// TIA Portal project "ForExportDB" (V14)

(* hardware
DEVICE "S7300/ET200M station_1"  S7-300 station
   slot 0: "Rail_0"  Rail  6ES7 390-1***0-0AA0
   slot 2: "PLC_1"  CPU 315-2 PN/DP  6ES7 315-2EH14-0AB0  V3.2
      slot 2: "PROFINET interface_1"  PN-IO
         slot 1: "Port_1"  Port
         slot 2: "Port_2"  Port
*)

// ===== PLC "PLC_1"  CPU 315-2 PN/DP =====

TYPE "UDT_DESCRETE_MODULE"
   STRUCT
      D_0 : Bool;
      D_1 : Bool;
      D_2 : Bool;
      D_3 : Bool;
      D_4 : Bool;
      D_5 : Bool;
      D_6 : Bool;
      D_7 : Bool;
      xEmpty : Bool;
      bByte : Byte;
   END_STRUCT;
END_TYPE

TYPE "UDT_FLOWRATE_PULSE"
   STRUCT
      iPulseCounter : Int;   // Счетчик импульсов
      xResetCounter : Bool;   // Сброс счетчика
      rPulseFlowRate : Real;   // Расход
      rPulseRes : Real := 100.0;   // Сколько мл/л на импульс (100 мл / имп)
      rSumFlowPanel : Real;   // Суммарный расход всего
      rSumFlowProg : Real;   // Суммарный расход доза
      xResetFlowRateProg : Bool;   // Сброс СРВ
      xResetFlowRatePanel : Bool;   // Сброс СРД
   END_STRUCT;
END_TYPE

TYPE "UDT_ALARM"
   STRUCT
      LAMPS : Struct   // Индикация
         Lamp1 : Struct   // Светофор 1
            rFlashTimer : Real := 3.0;   // Значение мигания
            iLampState : Array[0..2] of Int;   // Режим работы ламп
            xLampFlash : Array[0..2] of Bool;   // Мигание включено или нет
            xLampSet : Array[0..2] of Bool;
         END_STRUCT;
         Lamp2 : Struct   // Светофор 2
            rFlashTimer : Real := 1.0;   // Значение мигания
            iLampState : Array[0..2] of Int;   // Режим работы ламп
            xLampFlash : Array[0..2] of Bool;   // Мигание включено или нет
            xLampSet : Array[0..2] of Bool;
         END_STRUCT;
         Panel : Struct   // Индикация на панели
            xBuzzer : Bool;   // Звук
            xStartLamp : Bool;   // Старт
            xStopLamp : Bool;   // Стоп
            xResetLamp : Bool;   // Сброс
         END_STRUCT;
         Stand : Struct   // Индикация на стенде
            xRunMotor : Bool;   // Лампа мотора
            rRunMotorFlashTime : Real := 2.0;   // Значение мигания
         END_STRUCT;
      END_STRUCT;
      STATUS : Struct   // Статусы
         xErrorCommon : Bool;   // Общая ошибка
         xWarningCommon : Bool;   // Общее предупреждение
         iWarning : Int;   // Слово состояние предупреждения
         iError : Int;   // Слово состояния ошибки
         bMode : Byte;   // Текущий режим работы системы 16#25-26-29-2A
      END_STRUCT;
   END_STRUCT;
   // LAMPS.Lamp1.xLampFlash[0] := TRUE;
   // LAMPS.Lamp1.xLampFlash[1] := TRUE;
   // LAMPS.Lamp1.xLampFlash[2] := TRUE;
   // LAMPS.Lamp2.xLampFlash[0] := FALSE;
   // LAMPS.Lamp2.xLampFlash[1] := TRUE;
   // LAMPS.Lamp2.xLampFlash[2] := FALSE;
   // LAMPS.Lamp1.iLampState[0] := 0;   // Режим работы ламп красный
   // LAMPS.Lamp1.iLampState[1] := 1;   // Режим работы ламп желтый
   // LAMPS.Lamp1.iLampState[2] := 2;   // Режим работы ламп зеленый
   // LAMPS.Lamp2.iLampState[0] := 2;   // Режим работы ламп красный
   // LAMPS.Lamp2.iLampState[1] := 1;   // Режим работы ламп желтый
   // LAMPS.Lamp2.iLampState[2] := 0;   // Режим работы ламп зеленый
END_TYPE

TYPE "UDT_ANALOG_AI_MODULE"
   STRUCT
      AI_0 : Struct
         RAW : "UDT_IO_ANALOG_M1";
         SCALE : "UDT_SCALE_AI";
      END_STRUCT;
      AI_1 : Struct
         RAW : "UDT_IO_ANALOG_M1";
         SCALE : "UDT_SCALE_AI";
      END_STRUCT;
      AI_2 : Struct
         RAW : "UDT_IO_ANALOG_M1";
         SCALE : "UDT_SCALE_AI";
      END_STRUCT;
      AI_3 : Struct
         RAW : "UDT_IO_ANALOG_M1";
         SCALE : "UDT_SCALE_AI";
      END_STRUCT;
   END_STRUCT;
END_TYPE

TYPE "UDT_UDM200_MB_REG"
   STRUCT
      iSave : Int := 0;   // Запись
      iMinFreq : Int := 0;   // Запись
      iMaxFreq : Int := 5000;   // Запись
      iSetSpeed : Int := 0;   // Запись
      iCurrLimit : Int := 1300;   // Запись
      iNomDriveCurr : Int := 65;   // Запись
      iNomDriveSpeed : Int := 26500;   // Запись
      iNomDriveVoltage : Int := 220;   // Запись
      iNomDriveFreq : Int := 5000;   // Запись
      iNomDrivePowerFreq : Int := 85;   // Запись
      iAutotuneSelect : Int := 0;   // Запись
      iControlModeSelect : Int := 1;   // Запись
      iControlWord : Int;   // Запись
      iDriveReset : Int;   // Запись
      iActualDriveCurr : Int;   // Чтение
      iActualDriveCurrLoad : Int;   // Чтение
      iDriveTempPerc : Int;   // Чтение
      iDriveLoadPerc : Int;   // Чтение
      iActualDriveFreq : Int;   // Чтение
      iActualDriveVoltage : Int;   // Чтение
      iActualDrivePower : Int;   // Чтение
      iActualDriveRPM : Int;   // Чтение
      iPowerCounter : Int;   // Чтение
      iDriveAnalogInput_1 : Int;   // Чтение
      iDriveAnalogInput_2 : Int;   // Чтение
      iTempPowerModule : Int;   // Чтение
      iTempAddModule : Int;   // Чтение
      iMagnetisingCurrent : Int;   // Чтение
      iStatusWordDrive : Int;   // Чтение
      iLastError : Int;   // Чтение
      iLoadWarning : Int;   // Чтение
      iHeatWarning : Int;   // Чтение
      iCommonWarning : Int;   // Чтение
      iStatusWordCon : Int;   // Чтение
      iControlWordEnable : Int := 1;   // Чтение/Запись
   END_STRUCT;
END_TYPE

TYPE "UDT_UDM200_MB_SYS"
   STRUCT
      UNIDRIVE_M200_ADDR : Struct   // Адреса регистров (откуда читать, куда записать)
         wADDR_WRITE : Word := 16#0;   // Адрес записи
         wADDR_READ_1 : Word := 16#D;   // Адрес чтения 1
         wADDR_READ_2 : Word := 16#17;   // Адрес чтения 2
         wADDR_RW : Word := 16#21;   // Адрес чтения/записи
      END_STRUCT;
      UNIDRIVE_M200_SYS : Struct   // Системные (длина запроса, адрес, команды)
         iLEN_WRITE : Int := 13;   // Сколько регистров записать
         iLEN_READ_1 : Int := 10;   // Сколько регистров считать 1
         iLEN_READ_2 : Int := 10;   // Сколько регистров считать2
         iLEN_READWRITE : Int := 1;   // Сколько считать/записать
         bSLAVE_ID : Byte := 16#A;   // Адрес устройства
         bMODE_MULT_WORDS_READ : Byte := 16#03;   // Команда чтение нескольких регистров
         bMODE_MULT_WORDS_WRITE : Byte := 16#10;   // Команда запись нескольких регистров
      END_STRUCT;
   END_STRUCT;
END_TYPE

TYPE "UDT_PID"
   STRUCT
      rSetValue : Real;   // SP
      rProcessVariable : Real;   // PV
      rOutput : Real;   // MV
      rKp : Real;   // П
      iKi : Int;   // И
      iKd : Int;   // Д
      rErrorValue : Real;   // SP-PV
      xOutputHigh : Bool;   // MV H
      xOutputLow : Bool;   // MV L
   END_STRUCT;
END_TYPE

TYPE "UDT_ANALOG_VALVE"
   STRUCT
      rMinOpenPerc : Real := 0.0;   // Минимальное значение открытия
      rMaxOpenPerc : Real := 100.0;   // Максимальное значение открытия
      rSetOpenPercMan : Real := 100.0;   // Уставка в ручном
      rSetOpenPerc : Real := 100.0;   // Откуда берем уставку
      rTimeToOpen : Real := 20.0;   // Время открытия клапана (HMI)
      xError : Bool;   // Общая ошибка
      xWarning : Bool;   // Общее предупреждение
      iAlarmC : Int;   // Код ошибки
      iSCADAState : Int;   // Состояние для скады
      xWork : Bool;
      xPause : Bool;
      xCmdOn : Bool;
      xFault : Bool;
      xCmdPermit : Bool;
      xGoRun : Bool;
   END_STRUCT;
END_TYPE

TYPE "UDT_PUMP"
   STRUCT
      iSetFreqMan : Int;   // Задание в ручном
      iSetFreq : Int;   // Принимает частоту и передает по МБ
      aiSetPumpCommandWord : Array[0..1] of Int;   // Список команд
      xGoRun : Bool;   // Принимает команды и передает по МБ
      xSpeedControlSelect : Bool := true;   // Выбор: задание скорости по МБ (1) или по аналог (0)
      rCurCosFI : Real;   // Текущий косинус
      iMaxFreq : Int := 5000;   // Макс частота (5000 = 50 Hz)
      iMinFreq : Int := 0;   // Мин частота
      iCurVoltage : Int;   // Напряжение на насосе (В)
      iCurCurrent : Int;   // Ток на моторе (А)
      iCurLoadPerc : Int;   // Нагрузка на моторе (%)
      rCurLoadValue : Real;   // Нагрузка на моторе (кВт)
      rSumLoad : Real;
      iCurFreq : Int;   // Текущая частота
      iCurModuleTemp : Int;   // Температура модуля
      iAlarmC : Int;   // Слово ошибка насоса
      xCmdOn : Bool;   // Команда на запуск из программ
      xWork : Bool;   // Насос запустился (с частотника)
      xTempError : Bool;   // Перегрев насоса
      xCosFIError : Bool;   // Сухой ход
      xCmdPermit : Bool;   // Разрешен запуск
      xPause : Bool;   // Насос ожидает
      xError : Bool;   // Общая ошибка
      xService : Bool;   // Сервис
      rOperTime : Real;   // Время наработки (мин)
      xResetOperTime : Bool;   // Сброс времени наработки
      xResetLoadSum : Bool;   // Сброс счетчика квт
      diTFHTimer : DInt;   // Таймер
      iTimeToRun : Int := 3;   // Время запуска (сек)
      iPLCState : Int;   // Состояние внутри программы
      iSCADAState : Int;   // Состояние для СКАДА
      xFault : Bool;   // Ошибка с реле (от частотника)
      iSetTemp : Int := 45;   // Уставка температуры
      iFlashTime : Int := 3;   // Время мигания лампы РАБОТА
      xTempErrorEnable : Bool;   // Активировать защиту от перегрева
      xCosFIProtectEnable : Bool;   // Автивировать защиту от сухого хода
      rSetCosFI : Real := 0.7;   // Уставка COSFI
      rCosFIProtectTime : Real := 10.0;   // Задержка на срабатываение защиты от сухого хода
      rTempErrorTime : Real := 5.0;   // Задержка на срабатываение защиты от перегрева
   END_STRUCT;
   // aiSetPumpCommandWord[0] := 0;   // СТОП
   // aiSetPumpCommandWord[1] := 387;   // ПУСК ВПЕРЕД
END_TYPE

TYPE "UDT_ANALOG_AO_MODULE"
   STRUCT
      AO_0 : Struct
         RAW : "UDT_IO_ANALOG_M1";
         SCALE : "UDT_SCALE_AO";
      END_STRUCT;
      AO_1 : Struct
         RAW : "UDT_IO_ANALOG_M1";
         SCALE : "UDT_SCALE_AO";
      END_STRUCT;
      AO_2 : Struct
         RAW : "UDT_IO_ANALOG_M1";
         SCALE : "UDT_SCALE_AO";
      END_STRUCT;
      AO_3 : Struct
         RAW : "UDT_IO_ANALOG_M1";
         SCALE : "UDT_SCALE_AO";
      END_STRUCT;
   END_STRUCT;
END_TYPE

TYPE "UDT_BUTTONS"
   STRUCT
      bSelectControlSB1 : Byte := 16#01;   // SELECT CONTROL: 0 - Idle, 1 - Man, 2 - Auto
      bSelectModeSB2 : Byte := 16#01;   // SELECT MODE: 0 - Idle, 1 - Discrete, 2 - Cont
      bSelectProcessSP1 : Byte := 16#01;   // SELECT PROCESS: 0 - idle, 1 - level / flow, 2 - level / dosing, 3 - temperature
      xStartSL1 : Bool;   // Старт кнопка
      xStartPanelSL1 : Bool;   // Старт с панели
      xStopSL2 : Bool;   // Стоп кнопка
      xStopPanelSL2 : Bool;   // Стоп с панели
      xEmergencyStopSL3 : Bool;   // EMERGENCY STOP
      xResetSL4 : Bool;   // Сброс кнопка (с панели)
      xAuto : Bool;   // Селектор Авто
      xMan : Bool;   // Селектор Ручн
      xSelectMode1 : Bool;   // Выбаран режим 1
      xSelectMode2 : Bool;   // Выбран режим 2
   END_STRUCT;
END_TYPE

TYPE "UDT_PIDCONTC"
   STRUCT
      xResetPID : Bool;   // Сброс ПИД
      xPVPerOn : Bool;   // Вход переферии (лог)
      xManControl : Bool;   // Ручной режим
      xP_ON : Bool := true;   // П вкл
      xI_ON : Bool := true;   // И вкл
      xD_ON : Bool := true;   // Д вкл
      xI_HOLD : Bool;   // Удержание И
      xI_ITL_HOLD : Bool;   // Удержание И
      rI_ITLVAL : Real;   // Значение И
      wPVPer : Word;   // Переферия вход
      tTimePIDCycle : Time := T#100ms;   // Время цикла ПИД
      rSetPoint : Real;   // Уставка
      rProcessVariable : Real;   // Обратная связь
      rManControlValue : Real;   // Значение в ручном режиме
      rK_p : Real;   // П
      tK_i : Time := T#5s;   // И
      tK_d : Time := T#5s;   // Д
      tK_d_lagtime : Time := T#1s;   // Время диф
      rDeadBandWidth : Real;   // Зона нечувствительности
      rLimitOutputH : Real := 100.0;   // Выход управляющий максимум
      rLimitOutputL : Real := 0.0;   // Выход управляющий минимум
      rPV_FAC : Real := 1.0;   // Инверсия значения с датчика
      rPV_OFFSET : Real;   // Сдвиг значения с датчика
      rLMN_FAC : Real;   // Инверсия выхода
      rLMN_OFFSET : Real;   // Сдвиг выхода (при инверсии 100)
      rDisturbVariable : Real;   // Возмущающее воздействие
      rPIDOutput : Real;   // Выход ПИД
      xOutputLimitH : Bool;   // Выход ПИД достиг максимума
      xOutputLimitL : Bool;   // Выход ПИД достиг минимума
      rOuputP : Real;   // П выход
      rOuputI : Real;   // И выход
      rOuputD : Real;   // Д выход
      rProcessVariableOutput : Real;   // Выход значения датчика
      rErrorSignalValue : Real;   // Ошибка рассогласования
      wReserv : Word;   // Резерв
   END_STRUCT;
END_TYPE

TYPE "UDT_ENERGYMETER"
   STRUCT
      L1_Voltage : Real;   // Напряжение фаза 1
      L2_Voltage : Real;   // Напряжение фаза 2
      L3_Voltage : Real;   // Напряжение фаза 3
      L1_Current : Real;   // Ток фаза 1
      L2_Current : Real;   // Ток фаза 2
      L3_Current : Real;   // Ток фаза 3
      Psum : Real;   // Суммарное потребление кВт
      Pcom : Real;   // Общее активное потребление кВт
      cosfi : Real;   // Косинус
      xError : Bool;   // Ошибка общая датчика
      xWarning : Bool;   // Предупреждение общее датчика
      iAlarmC : Int;   // Код ошибки
      iSCADAState : Int;   // Код состояния
      rSetVoltageL1 : Real := 220.0;
      rSetCurL1 : Real := 15.0;
      rSetCosFIL1 : Real := 0.5;
      rSetDeltaVoltage : Real;
      rSetDeltaCurrent : Real;
      rSetDeltaCosFI : Real;
      DPRD_RET_VAL : Int;   // Буфер
      DPWR_RET_VAL : Int;   // Буфер
   END_STRUCT;
END_TYPE

TYPE "UDT_ANALOG_SENSOR"
   STRUCT
      Raw : Real;   // Значение токового сигнала
      Scale : Real;   // Значение масштабированного сигнала
      Perc : Real;   // Значение в процентах
      xError : Bool;   // Общая ошибка
      xWarning : Bool;   // Общее предупреждение
      iAlarmC : Int;   // Код ошибки
      iSCADAState : Int;   // Сотояние для скады
      iTimeToError : Int;   // Задержка на выдачу ошибки
      rHighSP : Real := 65.0;
      rLowSP : Real := 5.0;
      iSPEnable : Int;   // 0 - нет, 1 - предупреждение, 2 - ошибка
   END_STRUCT;
END_TYPE

// folder: EnergyMeter

TYPE "EM_DATA_R1"
TITLE = UDT Function block to control a SLIO energy counter module
// #CurrentVersion = 2.0.0
   STRUCT
      HEADER : Struct   // Additional info: Status Global 0x41=Init Busy/0x42=Init Done/0xC0 Init Error
         Timeout : Time := T#5S;   // Input: Timeout value for internal command interface
         Polltime : Time := T#1S;   // Input: Time interval for periodically reading
         Control_Global : Byte := BYTE#16#01;   // Input: Bit0=Read values periodically/ Bit1=Read values once/ Bit7=Init Block
         Status_Global : Byte;   // Output: 0x00=never executed/0x01=Busy/0x02=Done/0x41,42,C0=Init /0x80=Error
         Status_Alarm_Global : Byte;   // Output: Error flags
         Cmd : Byte;   // Input: Bit0=Reset en val./ Bit1=Reset transducer/ Bit2=Reset alarms / Bit3=Write en val.
         Status_Cmd : Byte;   // Output: 0x00=never executed/ 0x01=Busy/ 0x02=Done/ 0x80=Error
         Jobtime : Time;   // Output: Time period for readout the measurement values or execute a command
         DsID : Byte;   // Output: Reference to data consistency of measurement values
         Frame_ID : Byte;   // Output: ID of currently read frame
         Error_ID : Word;   // Output: Error information
         Status_ReadVersion : Byte;   // Output: 0x00=never executed/ 0x01=Busy/ 0x02=Done/ 0x80=Error
         Reserve : Array[1..15] of Byte;   // Static: Reserve for future expansions
      END_STRUCT;
      VersionInfo : Struct   // Firmware version information
         FirmwareMajor : Byte;   // Output: Firmware major verion
         FirmwareMinor : Byte;   // Output: Firmware minor version
         FirmwareRevision : Byte;   // Output: Firmware revision
         ProtocollMajor : Byte;   // Output: Protocoll major version
         ProtocollMinor : Byte;   // Output: Protocoll minor version
         ProtocollRevision : Byte;   // Output: Protocoll revision
         ChipDateYear : Word;   // Output: Year of measurement chip
         ChipDateMonth : Byte;   // Output: Month of measurement chip
         ChipDateDay : Byte;   // Output: Day of measurement chip
      END_STRUCT;
      ACTIVE_EN_CONSUMED : Struct   // ID1=Active energy consumed: UINT32, 1Wh
         Read_Mode : Byte := BYTE#16#01;   // Input: Bit0=Measurement value is read
         Value : DWord;   // Output: Measurement value
      END_STRUCT;
      ACTIVE_EN_DELIVERED : Struct   // ID2=Active energy delivered: UINT32, 1Wh
         Read_Mode : Byte := BYTE#16#01;   // Input: Bit0=Measurement value is read
         Value : DWord;   // Output: Measurement value
      END_STRUCT;
      ACTIVE_EN_L1_CONSUMED : Struct   // ID3=Active energy phase1 consumed: UINT32, 1Wh
         Read_Mode : Byte := BYTE#16#01;   // Input: Bit0=Measurement value is read
         Value : DWord;   // Output: Measurement value
      END_STRUCT;
      ACTIVE_EN_L1_DELIVERED : Struct   // ID4=Active energy phase1 delivered: UINT32, 1Wh
         Read_Mode : Byte := BYTE#16#01;   // Input: Bit0=Measurement value is read
         Value : DWord;   // Output: Measurement value
      END_STRUCT;
      ACTIVE_EN_L2_CONSUMED : Struct   // ID5=Active energy phase2 consumed: UINT32, 1Wh
         Read_Mode : Byte := BYTE#16#01;   // Input: Bit0=Measurement value is read
         Value : DWord;   // Output: Measurement value
      END_STRUCT;
      ACTIVE_EN_L2_DELIVERED : Struct   // ID6=Active energy phase2 delivered: UINT32, 1Wh
         Read_Mode : Byte := BYTE#16#01;   // Input: Bit0=Measurement value is read
         Value : DWord;   // Output: Measurement value
      END_STRUCT;
      ACTIVE_EN_L3_CONSUMED : Struct   // ID7=Active energy phase3 consumed: UINT32, 1Wh
         Read_Mode : Byte := BYTE#16#01;   // Input: Bit0=Measurement value is read
         Value : DWord;   // Output: Measurement value
      END_STRUCT;
      ACTIVE_EN_L3_DELIVERED : Struct   // ID8=Active energy phase3 delivered: UINT32, 1Wh
         Read_Mode : Byte := BYTE#16#01;   // Input: Bit0=Measurement value is read
         Value : DWord;   // Output: Measurement value
      END_STRUCT;
      TOTAL_ACTIVE_POWER : Struct   // ID9=Total active power: UINT32, 1mW
         Read_Mode : Byte := BYTE#16#01;   // Input: Bit0=Measurement value is read
         Value : DWord;   // Output: Measurement value
      END_STRUCT;
      TOTAL_REACTIVE_POWER : Struct   // ID10=Total reactive power: INT32, 1mW
         Read_Mode : Byte := BYTE#16#01;   // Input: Bit0=Measurement value is read
         Value : DWord;   // Output: Measurement value
      END_STRUCT;
      TOTAL_APPARENT_POWER : Struct   // ID11=Total apparent power: INT32, 1mW
         Read_Mode : Byte := BYTE#16#01;   // Input: Bit0=Measurement value is read
         Value : DWord;   // Output: Measurement value
      END_STRUCT;
      FREQUENCY : Struct   // ID12=Frequency: UINT16, 0.01Hz
         Read_Mode : Byte := BYTE#16#01;   // Input: Bit0=Measurement value is read
         Value : DWord;   // Output: Measurement value
      END_STRUCT;
      TOTAL_COS_PHI : Struct   // ID13=Total cos phi: INT8, 0.01
         Read_Mode : Byte := BYTE#16#01;   // Input: Bit0=Measurement value is read
         Value : DWord;   // Output: Measurement value
      END_STRUCT;
      TEMPERATURE : Struct   // ID14=Temperature: INT16, 0.01°C
         Read_Mode : Byte := BYTE#16#01;   // Input: Bit0=Measurement value is read
         Value : DWord;   // Output: Measurement value
      END_STRUCT;
      L1_ACTIVE_POWER : Struct   // ID15=Phase1 active power: INT32, 1mW
         Read_Mode : Byte := BYTE#16#01;   // Input: Bit0=Measurement value is read
         Value : DWord;   // Output: Measurement value
      END_STRUCT;
      L1_REACTIVE_POWER : Struct   // ID16=Phase1 reactive power: INT32, 1mW
         Read_Mode : Byte := BYTE#16#01;   // Input: Bit0=Measurement value is read
         Value : DWord;   // Output: Measurement value
      END_STRUCT;
      L1_APPARENT_POWER : Struct   // ID17=Phase1 apparent power: INT32, 1mW
         Read_Mode : Byte := BYTE#16#01;   // Input: Bit0=Measurement value is read
         Value : DWord;   // Output: Measurement value
      END_STRUCT;
      L1_VOLTAGE : Struct   // ID18=Phase1 voltage: UINT32, 1mV
         Read_Mode : Byte := BYTE#16#01;   // Input: Bit0=Measurement value is read
         Value : DWord;   // Output: Measurement value
      END_STRUCT;
      L1_CURRENT : Struct   // ID19=Phase1 current: UINT32, 1mA
         Read_Mode : Byte := BYTE#16#01;   // Input: Bit0=Measurement value is read
         Value : DWord;   // Output: Measurement value
      END_STRUCT;
      L1_COS_PHI : Struct   // ID20=Phase1 cos phi: INT8, 0.01
         Read_Mode : Byte := BYTE#16#01;   // Input: Bit0=Measurement value is read
         Value : DWord;   // Output: Measurement value
      END_STRUCT;
      L1_HARMONIC_VOLTAGE : Struct   // ID21=Phase1 harmonic voltage: UINT32, 1mV
         Read_Mode : Byte := BYTE#16#01;   // Input: Bit0=Measurement value is read
         Value : DWord;   // Output: Measurement value
      END_STRUCT;
      L1_HARMONIC_CURRENT : Struct   // ID22=Phase1 harmonic current: UINT32, 1mA
         Read_Mode : Byte := BYTE#16#01;   // Input: Bit0=Measurement value is read
         Value : DWord;   // Output: Measurement value
      END_STRUCT;
      L2_ACTIVE_POWER : Struct   // ID23=Phase2 active power: UINT32, 1mW
         Read_Mode : Byte := BYTE#16#01;   // Input: Bit0=Measurement value is read
         Value : DWord;   // Output: Measurement value
      END_STRUCT;
      L2_REACTIVE_POWER : Struct   // ID24=Phase2 reactive power: UINT32, 1mW
         Read_Mode : Byte := BYTE#16#01;   // Input: Bit0=Measurement value is read
         Value : DWord;   // Output: Measurement value
      END_STRUCT;
      L2_APPARENT_POWER : Struct   // ID25=Phase2 apparent power: UINT32, 1mW
         Read_Mode : Byte := BYTE#16#01;   // Input: Bit0=Measurement value is read
         Value : DWord;   // Output: Measurement value
      END_STRUCT;
      L2_VOLTAGE : Struct   // ID26=Phase2 voltage: UINT32, 1mV
         Read_Mode : Byte := BYTE#16#01;   // Input: Bit0=Measurement value is read
         Value : DWord;   // Output: Measurement value
      END_STRUCT;
      L2_CURRENT : Struct   // ID27=Phase2 current: UINT32, 1mA
         Read_Mode : Byte := BYTE#16#01;   // Input: Bit0=Measurement value is read
         Value : DWord;   // Output: Measurement value
      END_STRUCT;
      L2_COS_PHI : Struct   // ID28=Phase2 cos phi: INT8, 0.01
         Read_Mode : Byte := BYTE#16#01;   // Input: Bit0=Measurement value is read
         Value : DWord;   // Output: Measurement value
      END_STRUCT;
      L2_HARMONIC_VOLTAGE : Struct   // ID29=Phase2 harmonic voltage: UINT32, 1mV
         Read_Mode : Byte := BYTE#16#01;   // Input: Bit0=Measurement value is read
         Value : DWord;   // Output: Measurement value
      END_STRUCT;
      L2_HARMONIC_CURRENT : Struct   // ID30=Phase2 harmonic current: UINT32, 1mA
         Read_Mode : Byte := BYTE#16#01;   // Input: Bit0=Measurement value is read
         Value : DWord;   // Output: Measurement value
      END_STRUCT;
      L3_ACTIVE_POWER : Struct   // ID31=Phase3 active power: UINT32, 1mW
         Read_Mode : Byte := BYTE#16#01;   // Input: Bit0=Measurement value is read
         Value : DWord;   // Output: Measurement value
      END_STRUCT;
      L3_REACTIVE_POWER : Struct   // ID32=Phase3 reactive power: UINT32, 1mW
         Read_Mode : Byte := BYTE#16#01;   // Input: Bit0=Measurement value is read
         Value : DWord;   // Output: Measurement value
      END_STRUCT;
      L3_APPARENT_POWER : Struct   // ID33=Phase3 apparent power: UINT32, 1mW
         Read_Mode : Byte := BYTE#16#01;   // Input: Bit0=Measurement value is read
         Value : DWord;   // Output: Measurement value
      END_STRUCT;
      L3_VOLTAGE : Struct   // ID34=Phase3 voltage: UINT32, 1mV
         Read_Mode : Byte := BYTE#16#01;   // Input: Bit0=Measurement value is read
         Value : DWord;   // Output: Measurement value
      END_STRUCT;
      L3_CURRENT : Struct   // ID35=Phase3 current: UINT32, 1mA
         Read_Mode : Byte := BYTE#16#01;   // Input: Bit0=Measurement value is read
         Value : DWord;   // Output: Measurement value
      END_STRUCT;
      L3_COS_PHI : Struct   // ID36=Phase3 cos phi: INT8, 0.01
         Read_Mode : Byte := BYTE#16#01;   // Input: Bit0=Measurement value is read
         Value : DWord;   // Output: Measurement value
      END_STRUCT;
      L3_HARMONIC_VOLTAGE : Struct   // ID37=Phase3 harmonic voltage: UINT32, 1mV
         Read_Mode : Byte := BYTE#16#01;   // Input: Bit0=Measurement value is read
         Value : DWord;   // Output: Measurement value
      END_STRUCT;
      L3_HARMONIC_CURRENT : Struct   // ID38=Phase3 harmonic current: UINT32, 1mA
         Read_Mode : Byte := BYTE#16#01;   // Input: Bit0=Measurement value is read
         Value : DWord;   // Output: Measurement value
      END_STRUCT;
      EXCESS_ACTIVE_EN_CONSUME : Struct   // ID39=Excess active energy consumed: UINT32
         Read_Mode : Byte := BYTE#16#01;   // Input: Bit0=Measurement value is read
         Value : DWord;   // Output: Measurement value
      END_STRUCT;
      EXCESS_ACTIVE_EN_DELIVER : Struct   // ID40=Excess active energy delivered: UINT32
         Read_Mode : Byte := BYTE#16#01;   // Input: Bit0=Measurement value is read
         Value : DWord;   // Output: Measurement value
      END_STRUCT;
      STATUS_BITS : Struct   // ID41=Status bits: UINT32
         Read_Mode : Byte := BYTE#16#01;   // Input: Bit0=Status flags are read
         Value : DWord;   // Output: Measurement value
      END_STRUCT;
      RESERVE_42 : Struct   // ID42
         Read_Mode : Byte;   // Input: Bit0=Status flags are read
         Value : DWord;   // Output: Measurement value
      END_STRUCT;
      RESERVE_43 : Struct   // ID43
         Read_Mode : Byte;   // Input: Bit0=Status flags are read
         Value : DWord;   // Output: Measurement value
      END_STRUCT;
      RESERVE_44 : Struct   // ID44
         Read_Mode : Byte;   // Input: Bit0=Status flags are read
         Value : DWord;   // Output: Measurement value
      END_STRUCT;
      RESERVE_45 : Struct   // ID45
         Read_Mode : Byte;   // Input: Bit0=Status flags are read
         Value : DWord;   // Output: Measurement value
      END_STRUCT;
      RESERVE_46 : Struct   // ID46
         Read_Mode : Byte;   // Input: Bit0=Status flags are read
         Value : DWord;   // Output: Measurement value
      END_STRUCT;
      RESERVE_47 : Struct   // ID47
         Read_Mode : Byte;   // Input: Bit0=Status flags are read
         Value : DWord;   // Output: Measurement value
      END_STRUCT;
      RESERVE_48 : Struct   // ID48
         Read_Mode : Byte;   // Input: Bit0=Status flags are read
         Value : DWord;   // Output: Measurement value
      END_STRUCT;
      RESERVE_49 : Struct   // ID49
         Read_Mode : Byte;   // Input: Bit0=Status flags are read
         Value : DWord;   // Output: Measurement value
      END_STRUCT;
      RESERVE_50 : Struct   // ID50
         Read_Mode : Byte;   // Input: Bit0=Status flags are read
         Value : DWord;   // Output: Measurement value
      END_STRUCT;
      RESERVE_51 : Struct   // ID51
         Read_Mode : Byte;   // Input: Bit0=Status flags are read
         Value : DWord;   // Output: Measurement value
      END_STRUCT;
      RESERVE_52 : Struct   // ID52
         Read_Mode : Byte;   // Input: Bit0=Status flags are read
         Value : DWord;   // Output: Measurement value
      END_STRUCT;
      RESERVE_53 : Struct   // ID53
         Read_Mode : Byte;   // Input: Bit0=Status flags are read
         Value : DWord;   // Output: Measurement value
      END_STRUCT;
      RESERVE_54 : Struct   // ID54
         Read_Mode : Byte;   // Input: Bit0=Status flags are read
         Value : DWord;   // Output: Measurement value
      END_STRUCT;
      RESERVE_55 : Struct   // ID55
         Read_Mode : Byte;   // Input: Bit0=Status flags are read
         Value : DWord;   // Output: Measurement value
      END_STRUCT;
      RESERVE_56 : Struct   // ID56
         Read_Mode : Byte;   // Input: Bit0=Status flags are read
         Value : DWord;   // Output: Measurement value
      END_STRUCT;
      RESERVE_57 : Struct   // ID57
         Read_Mode : Byte;   // Input: Bit0=Status flags are read
         Value : DWord;   // Output: Measurement value
      END_STRUCT;
      RESERVE_58 : Struct   // ID58
         Read_Mode : Byte;   // Input: Bit0=Status flags are read
         Value : DWord;   // Output: Measurement value
      END_STRUCT;
      RESERVE_59 : Struct   // ID59
         Read_Mode : Byte;   // Input: Bit0=Status flags are read
         Value : DWord;   // Output: Measurement value
      END_STRUCT;
      RESERVE_60 : Struct   // ID60
         Read_Mode : Byte;   // Input: Bit0=Status flags are read
         Value : DWord;   // Output: Measurement value
      END_STRUCT;
      SetValues : Struct   // Setvalues for
         EN_L1_CONSUMED : DWord;   // Input: Setvalue for: ID3=Active energy phase1 consumed: UINT32, 1Wh
         EN_L1_DELIVERED : DWord;   // Input: Setvalue for: ID4=Active energy phase1 delivered: UINT32, 1Wh
         EN_L2_CONSUMED : DWord;   // Input: Setvalue for: ID5=Active energy phase2 consumed: UINT32, 1Wh
         EN_L2_DELIVERED : DWord;   // Input: Setvalue for: ID6=Active energy phase2 delivered: UINT32, 1Wh
         EN_L3_CONSUMED : DWord;   // Input: Setvalue for: ID7=Active energy phase3 consumed: UINT32, 1Wh
         EN_L3_DELIVERED : DWord;   // Input: Setvalue for: ID8=Active energy phase3 delivered: UINT32, 1Wh
         EXCESS_ACTIVE_EN_CONSUME : DWord;   // Input: Setvalue for: ID40=Excess active energy consumed: UINT32
         EXCESS_ACTIVE_EN_DELIVER : DWord;   // Input: Setvalue for: ID39=Excess active energy delivered: UINT32
      END_STRUCT;
   END_STRUCT;
END_TYPE

TYPE "UDT_MB_SEND_RECV"
VERSION : 0.1
   STRUCT
      SEND_TGM : Array[0..9] of Byte;
      RECV_TGM : Array[0..9] of Byte;
   END_STRUCT;
END_TYPE

// folder: LeoFunc

TYPE "UDT_SCALE_AI"
VERSION : 0.1
   STRUCT
      VALUE : Real;   // Значение
      MAX_V : Real := 9999.0;   // Макс. масштаб величины
      MIN_V : Real;   // Мин. масштаб величины
      MAX_S : Real := 20.0;   // Макс. масштаб сигнала
      MIN_S : Real := 4.0;   // Мин. масштаб сигнала
   END_STRUCT;
END_TYPE

TYPE "UDT_IO_ANALOG_M1"
VERSION : 0.1
   STRUCT
      HW : Int;   // Единицы PLC
      CURR : Real;   // Ток, напряжение, сопротивление
      OUT : Real;   // Выход
   END_STRUCT;
END_TYPE

TYPE "UDT_SCALE_AO"
VERSION : 0.1
   STRUCT
      VALUE : Real;   // Значение
      MAX_V : Real := 100.0;   // Макс. масштаб величины
      MIN_V : Real := 0.0;   // Мин. масштаб величины
      MAX_S : Real := 20.0;   // Макс. масштаб сигнала
      MIN_S : Real := 4.0;   // Мин. масштаб сигнала
   END_STRUCT;
END_TYPE

// folder: (top level)

DATA_BLOCK "SCADA_DATA"   // DB10
{ S7_Optimized_Access := 'FALSE' }
VERSION : 0.1
   VAR
      BTN_SW : "UDT_BUTTONS";   // Кнопки
      ALARM_SETTINGS : "UDT_ALARM";   // Световая индикация и статусы
      SENSORS : Struct   // Датчики
         FLOWMETER : Struct   // FQ1 расходомер
            FQ1 : "UDT_ANALOG_SENSOR";
            rSumFlowAll : Real;   // Расход всего
            rSumFlowDose : Real;   // Расход за дозу
         END_STRUCT;
         L1 : "UDT_ANALOG_SENSOR";   // Датчик уровня Т1
         L2 : "UDT_ANALOG_SENSOR";   // Датчик уровня Т2
         POT : "UDT_ANALOG_SENSOR";   // Потенциометр
         ENERGYMETER : "UDT_ENERGYMETER";   // Модуль электроэнергии
      END_STRUCT;
      MECH : Struct   // Исполнительные механизмы
         VALVES : Struct   // Клапана
            HV1 : "UDT_ANALOG_VALVE";   // Клапан HV1
            HV2 : "UDT_ANALOG_VALVE";   // Клапан HV2
         END_STRUCT;
         PUMPS : Struct   // Насосы
            M1 : "UDT_PUMP";   // Насос М1
         END_STRUCT;
      END_STRUCT;
      PROCESS : Struct   // Процессы
         LEVELDOSE_SETTINGS : Struct   // Процесс дозирования и регулирования уровня
            rSetDoseVolume : Real := 8.0;   // Размер дозы (л)
            iCurDose : Int;   // Номер текущей дозы
            rMinLevel_T2 : Real := 15.0;   // Минимальный уровень Т2
            rMaxLevel_T2 : Real := 30.0;   // Максимальный уровень Т2
            iSetDoseCount : Int := 3;   // Уставка количества доз
            rSetTimeInterval : Real := 15.0;   // Уставка времени между дозами
            iProcessState : Int;   // Состояние процесса
            rTimeDelayMinLevel : Real := 3.0;   // Время задержки выключения насоса
            rTimeUntilNextDose : Real;   // Текущее время до следующей дозы
            rTimePausedFill : Real;   // Текущее время паузы при наполнении Т2
            PID_HV2_LEVEL_T2_SETTINGS : "UDT_PID";   // ПИД регулятор уровня Т2 клапаном HV2
         END_STRUCT;
         LEVELFLOW_SETTINGS : Struct   // Процесс регулирования расход и уровень
            iSelectPID : Int := 1;   // Выбор ПИД (0 - насос, 1 - клапан)
            PID_FLOW_T2_CASCADE : Struct   // ПИД контур регулирования Т2 HV2
               PID_MASTER : "UDT_PID";   // Мастер
               PID_SLAVE : "UDT_PID";   // Слейв
            END_STRUCT;
            PID_HV1_FLOW_T2_SETTINGS : "UDT_PID";   // ПИД расход HV1
            PID_M1_FLOW_T2_SETTINGS : "UDT_PID";   // ПИД расход M1
            PID_HV1_LEVEL_T1_SETTINGS : "UDT_PID";   // ПИД уровень Т1 HV1
            PID_M1_LEVEL_T1_SETTINGS : "UDT_PID";   // ПИД уровень Т1 M1
            rSetLevelT1 : Real := 25.0;
            rSetFlowRate : Real := 8.0;
            rSetLevelT2 : Real := 30.0;
         END_STRUCT;
         OTHER_SETTINGS : Struct   // Дополнительные настройки
            rT1_H : Real := 0.05;   // Уровень Т1
            rT1_L : Real;
            rT2_H : Real := 0.05;   // Уровень Т2
            rT2_L : Real;
            xMinLevel_T2 : Bool;
            xMaxLevel_T2 : Bool;
            xMinLevel_T1 : Bool;
            xMaxLevel_T1 : Bool;
            xEnableProtectT2 : Bool := true;
         END_STRUCT;
      END_STRUCT;
      MODBUS : Struct
         UNIDRIVE_M200 : Struct
            iCurQueryTime : Int;
            iCurQueryNum : Int;
            iLastQueryError : Int;
            bSlaveAddress : Byte := 16#A;
            iAlarmC : Int;
            iSCADAState : Int;
            xError : Bool;
         END_STRUCT;
      END_STRUCT;
      PLC_COUNTER : Int;
   END_VAR
BEGIN
   PROCESS.LEVELDOSE_SETTINGS.PID_HV2_LEVEL_T2_SETTINGS.rSetValue := 25.0;
   PROCESS.LEVELDOSE_SETTINGS.PID_HV2_LEVEL_T2_SETTINGS.rKp := 15.0;
   PROCESS.LEVELDOSE_SETTINGS.PID_HV2_LEVEL_T2_SETTINGS.iKi := 30;
   PROCESS.LEVELDOSE_SETTINGS.PID_HV2_LEVEL_T2_SETTINGS.iKd := 8;
   MECH.VALVES.HV2.rMinOpenPerc := 0.0;
   PROCESS.LEVELFLOW_SETTINGS.PID_FLOW_T2_CASCADE.PID_MASTER.rKp := 28.5;
   PROCESS.LEVELFLOW_SETTINGS.PID_FLOW_T2_CASCADE.PID_MASTER.iKi := 2;
   PROCESS.LEVELFLOW_SETTINGS.PID_FLOW_T2_CASCADE.PID_MASTER.iKd := 34;
   MECH.VALVES.HV1.rMinOpenPerc := 25.0;
   PROCESS.LEVELFLOW_SETTINGS.PID_FLOW_T2_CASCADE.PID_SLAVE.rKp := 9.0;
   PROCESS.LEVELFLOW_SETTINGS.PID_FLOW_T2_CASCADE.PID_SLAVE.iKi := 45;
   PROCESS.LEVELFLOW_SETTINGS.PID_FLOW_T2_CASCADE.PID_SLAVE.iKd := 16;
   PROCESS.LEVELFLOW_SETTINGS.PID_HV1_FLOW_T2_SETTINGS.rKp := 3.7;
   PROCESS.LEVELFLOW_SETTINGS.PID_HV1_FLOW_T2_SETTINGS.iKi := 5;
   PROCESS.LEVELFLOW_SETTINGS.PID_HV1_FLOW_T2_SETTINGS.iKd := 2;
   PROCESS.LEVELFLOW_SETTINGS.PID_M1_FLOW_T2_SETTINGS.rKp := 3.7;
   PROCESS.LEVELFLOW_SETTINGS.PID_M1_FLOW_T2_SETTINGS.iKi := 5;
   PROCESS.LEVELFLOW_SETTINGS.PID_M1_FLOW_T2_SETTINGS.iKd := 0;
   PROCESS.LEVELFLOW_SETTINGS.PID_HV1_LEVEL_T1_SETTINGS.rKp := 24.0;
   PROCESS.LEVELFLOW_SETTINGS.PID_HV1_LEVEL_T1_SETTINGS.iKi := 20;
   PROCESS.LEVELFLOW_SETTINGS.PID_HV1_LEVEL_T1_SETTINGS.iKd := 2;
   PROCESS.LEVELFLOW_SETTINGS.PID_M1_LEVEL_T1_SETTINGS.rKp := 2.5;
   PROCESS.LEVELFLOW_SETTINGS.PID_M1_LEVEL_T1_SETTINGS.iKi := 3;
   MECH.PUMPS.M1.xTempErrorEnable := true;
   MECH.PUMPS.M1.xCosFIProtectEnable := true;
   MECH.PUMPS.M1.rCosFIProtectTime := 1.0;
   MECH.PUMPS.M1.rTempErrorTime := 15.0;
   MECH.PUMPS.M1.rSetCosFI := 0.125;
   MECH.VALVES.HV1.rTimeToOpen := 75.0;
   MECH.VALVES.HV2.rTimeToOpen := 75.0;
   SENSORS.ENERGYMETER.rSetVoltageL1 := 200.0;
   // ALARM_SETTINGS.LAMPS : Лампы
   // ALARM_SETTINGS.STATUS : Состояния
END_DATA_BLOCK

ORGANIZATION_BLOCK "Main"   // OB1, LAD
TITLE = "Main Program Sweep (Cycle)"
{ S7_Optimized_Access := 'FALSE' }
VERSION : 0.1
   VAR_TEMP
      OB1_EV_CLASS : Byte;   // Bits 0-3 = 1 (Coming event), Bits 4-7 = 1 (Event class 1)
      OB1_SCAN_1 : Byte;   // 1 (Cold restart scan 1 of OB 1), 3 (Scan 2-n of OB 1)
      OB1_PRIORITY : Byte;   // Priority of OB Execution
      OB1_OB_NUMBR : Byte;   // 1 (Organization block 1, OB1)
      OB1_RESERVED_1 : Byte;   // Reserved for system
      OB1_RESERVED_2 : Byte;   // Reserved for system
      OB1_PREV_CYCLE : Int;   // Cycle time of previous OB1 scan (milliseconds)
      OB1_MIN_CYCLE : Int;   // Minimum cycle time of OB1 (milliseconds)
      OB1_MAX_CYCLE : Int;   // Maximum cycle time of OB1 (milliseconds)
      OB1_DATE_TIME : Date_And_Time;   // Date and time OB1 started
   END_VAR
BEGIN
END_ORGANIZATION_BLOCK